// TwinCAT 3 PLC project T3TckitUtils_Plc
// Title: T3TckitUtils_Plc
// Company: Tc3 Project
// ProjectVersion: 1.0.0.0
// ProgramVersion: 3.1.4026.22
// libraries:
//   Tc2_Standard, * (Beckhoff Automation GmbH)
//   Tc2_System, * (Beckhoff Automation GmbH)
// project tree:
//   / PlcTask.TcTTO
//   POUs/ MAIN.TcPOU
//   POUs/PID/ FB_Pid.TcPOU, I_Pid.TcIO
//   POUs/RingBuffer/ FB_RingBuffer.TcPOU
//   POUs/Strings/ FB_StringBuilder.TcPOU, F_Contains.TcPOU, F_EndsWith.TcPOU, F_StartsWith.TcPOU, F_Trim.TcPOU
// real-time tasks:
//   TASK PlcTask: cycle T#10ms, priority 20, ADS port 350

CONFIGURATION T3TckitUtils_Plc
    RESOURCE PLC ON TwinCAT3
        TASK PlcTask(INTERVAL := T#10ms, PRIORITY := 20);
        PROGRAM MAIN WITH PlcTask : MAIN;
    END_RESOURCE
END_CONFIGURATION

// ---- POUs/PID/I_Pid.TcIO
INTERFACE I_Pid

METHOD Reset
END_METHOD

METHOD Update : LREAL
VAR_INPUT
    setpoint    : LREAL;
    measurement : LREAL;
    deltaT      : LREAL;
END_VAR
END_METHOD

END_INTERFACE

// ---- POUs/MAIN.TcPOU
PROGRAM MAIN
VAR
END_VAR

END_PROGRAM

// ---- POUs/PID/FB_Pid.TcPOU
FUNCTION_BLOCK FB_Pid
VAR
END_VAR

END_FUNCTION_BLOCK

// ---- POUs/RingBuffer/FB_RingBuffer.TcPOU
FUNCTION_BLOCK FB_RingBuffer
VAR
END_VAR

END_FUNCTION_BLOCK

// ---- POUs/Strings/FB_StringBuilder.TcPOU
FUNCTION_BLOCK FB_StringBuilder
VAR
END_VAR

END_FUNCTION_BLOCK

// ---- POUs/Strings/F_Contains.TcPOU
FUNCTION F_Contains : BOOL
VAR_INPUT
    s      : STRING;
    needle : STRING;
END_VAR

END_FUNCTION

// ---- POUs/Strings/F_EndsWith.TcPOU
FUNCTION F_EndsWith : BOOL
VAR_INPUT
    s      : STRING;
    suffix : STRING;
END_VAR

END_FUNCTION

// ---- POUs/Strings/F_StartsWith.TcPOU
FUNCTION F_StartsWith : BOOL
VAR_INPUT
    s      : STRING;
    prefix : STRING;
END_VAR

END_FUNCTION

// ---- POUs/Strings/F_Trim.TcPOU
FUNCTION F_Trim : STRING
VAR_INPUT
    s : STRING;
END_VAR

END_FUNCTION
